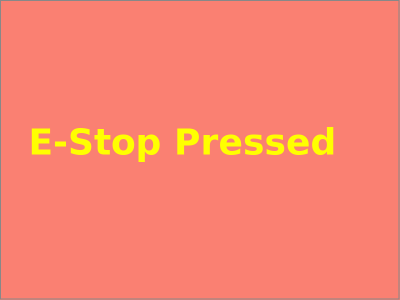
VISUALIZATION Dialog_Estop  // 400x300
    Label (31,79 303x126), "E-Stop Pressed"
END_VISUALIZATION

(* stored: Version 1.1.0.1, ProductVersion 3.1.4024.3
   Visu Dialog_Estop: Id {c6e79852-dd9a-42c3-8d32-1c6606b748d8} *)
